FUNCTION_BLOCK PUBLIC PAEThermometer EXTENDS PAESensorAnalog
VAR_INPUT
END_VAR
VAR_OUTPUT
END_VAR
VAR
END_VAR

END_FUNCTION_BLOCK

(* stored: Version 1.1.0.1, ProductVersion 3.1.4020.6
   POU PAEThermometer: Id {8fbdb98c-1add-4f79-a837-c916be146392}, SpecialFunc None *)
